{attribute 'Tc2GvlVarNames'}
VAR_GLOBAL


	R_BTN_S3: BOOL;



END_VAR

(* stored: Version 1.1.0.1, ProductVersion 3.1.0.26
   GVL Global_Constantes: Id {e69359d1-77c4-4d7b-aacc-c56c2e4d46f7} *)
